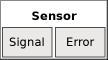
VISUALIZATION vSensorFrame  // 108x60
VAR_INPUT
		iNameIndex :INT;
END_VAR
VAR_IN_OUT
	fbSensor :FB_Sensor;

END_VAR
    Rectangle (0,0 108x60)
    Rectangle (2,27 50x30), "Signal", colour toggle: fbSensor.bSensorSignal
    Rectangle (55,27 50x30), "Error", colour toggle: fbSensor.prSensorOnError OR fbSensor.prSensorOffError
    Rectangle (3,1 102x30), "Sensor", text list: 'tlDevices', text index: iNameIndex
END_VISUALIZATION

(* stored: Version 1.1.0.1, ProductVersion 3.1.4024.15
   Visu vSensorFrame: Id {cbf39ea4-9e6c-4591-ada2-89e11b647e28} *)
